{attribute 'qualified_only'}
{attribute 'strict'}
TYPE E_SIGNAL :
(
	//periodic signals
	SINUS 		:= 1,
	COSINUS		:= 2,
	SQUARE		:= 3,
	TRIANGLE	:= 4,
	SAWTOOTH	:= 5,
	DIRAC_DELTA	:= 6,
	
	//discontinuous function
	SINGLE_DD	:= 7,	//single dirac delta
	STEP		:= 8,
	
	
	//other
	CONST 		:= 9,
	GAUSS_FUNC	:= 10,
	SINC		:= 11		
);
END_TYPE

(* stored: Version 1.1.0.1, ProductVersion 3.1.4024.4
   DUT E_SIGNAL: Id {f0806bfc-7f05-44e0-9957-8ac01948fdcf} *)
